Universal Robots PolyScope program: test_socket.urp

Program test_socket (installation=default directory=/programs/usbdisk createdIn=5.9.4.1031232 lastSavedIn=3.14.3.1031232 robotSerialNumber=2017332543)
Calibrated DH parameters: a=[0.000031, -0.243823, -0.204309, 0.000009, -0.000019, 0]; d=[0.152052, 0.291789, 9.837334, -10.016486, 0.085275, 0.082255]; alpha=[1.569617, -0.005691, 0.006147, 1.57048, -1.570017, 0]; deltaTheta=[-0.000062, -0.006867, 0.302677, -0.295865, 0.000039, 0.000042]
BeforeStart
  Loop While (checkContinuously=false) expression=not socket_open("192.168.2.130",50002)
    Wait Sleep waitTime=0.05
  data := socket_read_ascii_float(6)
  If to_str(data[1])≟"nan"
    Script: socket_close()
    Halt
  desired_q := [data[1], data[2], data[3], data[4], data[5], data[6]]
  MoveJ speed 30 deg/s, acceleration 40 deg/s^2 (useActiveTCP=true)
    Waypoint Waypoint (Variable): variable=desired_q
  Wait Sleep waitTime=0.5
  temp := get_actual_joint_positions()
  Loop Counting (count=6) loopVariable(name=Loop_2)
    var_1 := temp[Loop_2]-desired_q[Loop_2]
    If var_1<0
      var_1 := -var_1
    If var_1> 0.001
      Script: socket_send_string("Posicion no alcanzada")
      Script: socket_close()
      Halt
  Script: socket_send_string("Ready")
  Wait Sleep waitTime=0.05
Robot Program (runOnlyOnce=false)
  data := socket_read_ascii_float(6)
  Script: socket_send_string(get_actual_joint_positions())
  If to_str(data[1])≟"nan"
    Script: socket_close()
    Halt
  desired_q := [data[1], data[2], data[3], data[4], data[5], data[6]]
Thread Thread_1 (runOnlyOnce=false)
  Script: servoj(desired_q,0,0,0.008,0.1,100)
